PROGRAM AutoMain
VAR

END_VAR
VAR // added by the converter: edge detectors and wires of the graphical bodies
    _w1, _w2, _w3 : BOOL;
END_VAR

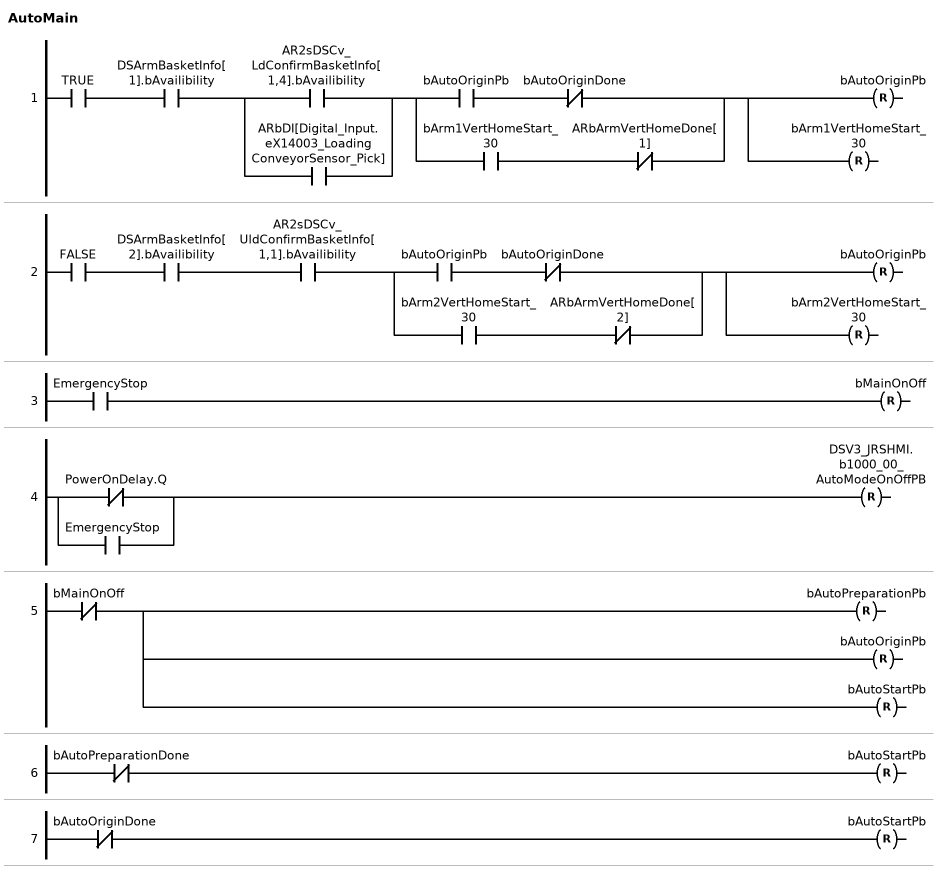
// NETWORK 1
_w1 := TRUE AND DSArmBasketInfo[1].bAvailibility AND (AR2sDSCv_LdConfirmBasketInfo[1,4].bAvailibility OR ARbDI[Digital_Input.eX14003_LoadingConveyorSensor_Pick]) AND (bAutoOriginPb AND NOT bAutoOriginDone OR bArm1VertHomeStart_30 AND NOT ARbArmVertHomeDone[1]);
bAutoOriginPb R= _w1;
bArm1VertHomeStart_30 R= _w1;

// NETWORK 2
_w2 := FALSE AND DSArmBasketInfo[2].bAvailibility AND AR2sDSCv_UldConfirmBasketInfo[1,1].bAvailibility AND (bAutoOriginPb AND NOT bAutoOriginDone OR bArm2VertHomeStart_30 AND NOT ARbArmVertHomeDone[2]);
bAutoOriginPb R= _w2;
bArm2VertHomeStart_30 R= _w2;

// NETWORK 3
bMainOnOff R= EmergencyStop;

// NETWORK 4
DSV3_JRSHMI.b1000_00_AutoModeOnOffPB R= NOT PowerOnDelay.Q OR EmergencyStop;

// NETWORK 5
_w3 := NOT bMainOnOff;
bAutoPreparationPb R= _w3;
bAutoOriginPb R= _w3;
bAutoStartPb R= _w3;

// NETWORK 6
bAutoStartPb R= NOT bAutoPreparationDone;

// NETWORK 7
bAutoStartPb R= NOT bAutoOriginDone;

END_PROGRAM

(* stored: Version 1.1.0.1, ProductVersion 3.1.4024.12
   POU AutoMain: Id {7deba789-5552-46b6-b0e5-c7cdc063d9b5}, SpecialFunc None *)
